(* CoDeSys 2.3 export: FTOGGLE.EXP *)

(* POU Fs/fToggle, ST *)
FUNCTION fToggle : BOOL
VAR_INPUT
	IN: BOOL;
END_VAR
IF IN THEN
	fToggle := FALSE;
ELSE
	fToggle := TRUE;
END_IF
END_FUNCTION
